FUNCTION_BLOCK FillPoly (* openCV fillPolygon *)
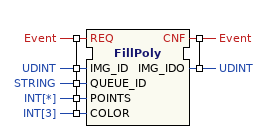
  EVENT_INPUT
    REQ WITH IMG_ID, QUEUE_ID, POINTS, COLOR;
  END_EVENT
  EVENT_OUTPUT
    CNF WITH IMG_IDO;
  END_EVENT
  VAR_INPUT
    IMG_ID : UDINT;
    QUEUE_ID : STRING;
    POINTS : ARRAY [*] OF INT;
    COLOR : ARRAY [0..2] OF INT;
  END_VAR
  VAR_OUTPUT
    IMG_IDO : UDINT;
  END_VAR
END_FUNCTION_BLOCK
